{attribute 'qualified_only'}
{attribute 'strict'}
TYPE E_SEEK_STYLE :
(
	E_STREAM_BEGIN := 0,
	E_STREAM_CURRENT,
	E_STREAM_END
);
END_TYPE

(* stored: Version 1.1.0.1, ProductVersion 3.1.4019.2
   DUT E_SEEK_STYLE: Id {b1b2c3c5-ec87-4c06-9d9d-6609942047fb} *)
